FUNCTION F_LogLA10C 
VAR_INPUT
	eLogLevel		: E_LogLevel;
	sLogger			: T_MaxString;
	sMessage		: T_MaxString;
	aArg1			: ANY;
	aArg2			: ANY;
	aArg3			: ANY;
	aArg4			: ANY;
	aArg5			: ANY;
	aArg6			: ANY;
	aArg7			: ANY;
	aArg8			: ANY;
	aArg9			: ANY;
	aArg10			: ANY;
	iContextBuilder	: I_ContextBuilder;
END_VAR

F_LogA(
	eLogLevel,
	sLogger,
	sMessage,
	10,
	aArg1,
	aArg2,
	aArg3,
	aArg4,
	aArg5,
	aArg6,
	aArg7,
	aArg8,
	aArg9,
	aArg10,
	iContextBuilder
);

END_FUNCTION

(* stored: Version 1.1.0.1, ProductVersion 3.1.4024.0
   POU F_LogLA10C: Id {30fb937e-6d33-4844-a5d7-58f0c98e875b}, SpecialFunc None *)
